// TIA Portal project "timers and counters" (V15.1)

(* hardware
DEVICE "S7-1200 station_1"  S7-1200 Station
   slot 0: "Rack_0"  S7-1200 Rack  Rack  V1.0
   slot 1: "PLC_1"  CPU 1212FC DC/DC/DC  6ES7 212-1AF40-0XB0  V4.2
*)

// ===== PLC "PLC_1"  CPU 1212FC DC/DC/DC =====

VAR_GLOBAL   // PLC tag table "Default tag table"
   "start" AT %I0.0 : Bool;
   "sensorb1" AT %I0.1 : Bool;
   "cylinder1" AT %Q0.0 : Bool;
   "waitled" AT %Q0.1 : Bool;
END_VAR

VAR_GLOBAL CONSTANT   // PLC tag table "Default tag table"
   "stamptime" : Time := T#4s;
   "waittime" : Time := T#20s;
   "countpart" : Int := 10;
END_VAR

// folder: System blocks/Program resources

DATA_BLOCK "IEC_Timer_0_DB_1"   // DB3
{ S7_Optimized_Access := 'TRUE' }
AUTHOR : Simatic
FAMILY : IEC
NAME : IEC_TMR
VERSION : 1.0
// stored: InstanceOfName IEC_TIMER
"IEC_TIMER"
BEGIN
END_DATA_BLOCK

DATA_BLOCK "IEC_Timer_0_DB_2"   // DB4
{ S7_Optimized_Access := 'TRUE' }
AUTHOR : Simatic
FAMILY : IEC
NAME : IEC_TMR
VERSION : 1.0
// stored: InstanceOfName IEC_TIMER
"IEC_TIMER"
BEGIN
END_DATA_BLOCK

DATA_BLOCK "IEC_Counter_0_DB_1"   // DB5
{ S7_Optimized_Access := 'TRUE' }
AUTHOR : Simatic
FAMILY : IEC
NAME : CNTR
VERSION : 1.0
// stored: InstanceOfName IEC_COUNTER
"IEC_COUNTER"
BEGIN
END_DATA_BLOCK

// folder: (top level)

ORGANIZATION_BLOCK "Main"   // OB1, LAD, ProgramCycle
TITLE = "Main Program Sweep (Cycle)"
{ S7_Optimized_Access := 'TRUE' }
VERSION : 0.1
BEGIN

REGION Network 1
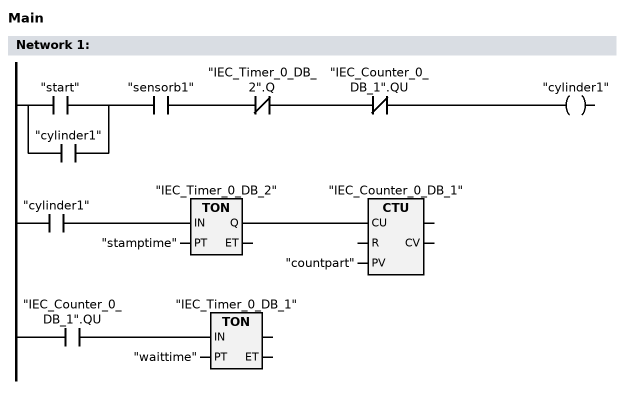
   "cylinder1" := ("start" OR "cylinder1") AND "sensorb1" AND NOT "IEC_Timer_0_DB_2".Q AND NOT "IEC_Counter_0_DB_1".QU;
   "IEC_Timer_0_DB_2".TON(IN := "cylinder1", PT := "stamptime");
   "IEC_Counter_0_DB_1".CTU(CU := "IEC_Timer_0_DB_2".Q, PV := "countpart");
   "IEC_Timer_0_DB_1".TON(IN := "IEC_Counter_0_DB_1".QU, PT := "waittime");
END_REGION
END_ORGANIZATION_BLOCK